TYPE ST_IdNode :
STRUCT
	nId : UINT;
	pNext : POINTER TO ST_IdNode;
END_STRUCT
END_TYPE

(* stored: Version 1.1.0.1, ProductVersion 3.1.4022.12
   DUT ST_IdNode: Id {7012813c-aefc-43a4-b66e-a6be4b08d383} *)
